PROGRAM SkillSet
VAR_INPUT
	Move_2P2			:Skill_Position_anfahren;
	Move_2P2_Advanced	:Skill_Position_anfahren_erweitert;
	
	Grip_2P2			:Skill_Greifer_Pos_Anfahren;
END_VAR

Move_2P2(
    Objekt := Anlage.UR5,
    eSysCommand := GVL.SystemCommand,
    eSysState := GVL.SystemState,
    eObjState := ANlage.UR5.P_State); // Skill_Position_anfahren
GVL.ErrorID := Move_2P2.iErrorID;
Grip_2P2(
    Objekt := Anlage.Gripper,
    eSysCommand := GVL.SystemCommand,
    eSysState := GVL.SystemState,
    eObjState := Anlage.Gripper.P_State); // Skill_Greifer_Pos_Anfahren
GVL.ErrorID := Grip_2P2.iErrorID;
Move_2P2_Advanced(
    Objekt := Anlage.UR5,
    eSysCommand := GVL.SystemCommand,
    eSysState := GVL.SystemState,
    eObjState := ANlage.UR5.P_State,
    sMessdaten := Anlage.HEX_E_V2.P_Messdaten); // Skill_Position_anfahren_erweitert
GVL.ErrorID := Move_2P2_Advanced.iErrorID;

END_PROGRAM

(* stored: Version 1.1.0.1
   POU SkillSet: Id {339b7e29-1078-4fc2-9977-078b023751ad}, SpecialFunc None *)
